TEXTLIST TL_PeersList
  0 = 'No peer'
  1 = 'Debug 1'
  2 = 'Debug 2'
  3 = 'Schneiden'
  4 = 'Umlenkung'
  5 = 'Bereitstellung'
  6 = 'Conveyor 1'
  7 = 'Conveyor 2'
  8 = 'Conveyor 3'
  9 = 'Conveyor 4'
  10 = 'Conveyor 5'
   = ''
END_TEXTLIST

(* stored: Version 1.1.0.1, ProductVersion 3.1.4022.16
   TextList TL_PeersList: Id {96e87d43-d769-433f-aea3-59627bba1876} *)
